// LS Electric XG5000 project: 0131 인버터 에스컬레이터
// PLC LSPLC

PROGRAM NewProgram (task: 스캔 프로그램)

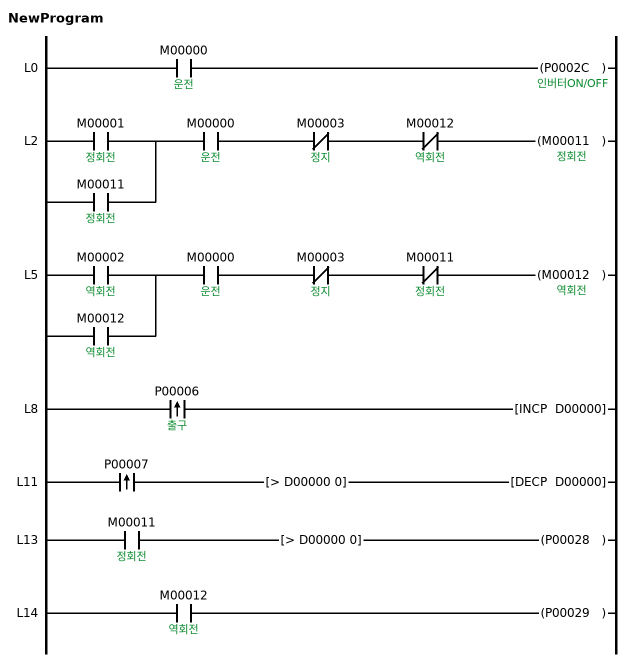
; L0
LOAD      M00000	// 운전
OUT       P0002C	// 인버터ON/OFF
; L2
LOAD      M00001	// 정회전
OR        M00011	// 정회전
AND       M00000	// 운전
AND NOT   M00003	// 정지
AND NOT   M00012	// 역회전
OUT       M00011	// 정회전
; L5
LOAD      M00002	// 역회전
OR        M00012	// 역회전
AND       M00000	// 운전
AND NOT   M00003	// 정지
AND NOT   M00011	// 정회전
OUT       M00012	// 역회전
; L8
LOADP     P00006	// 출구
INCP      D00000
; L11
LOADP     P00007
AND>      D00000 0
DECP      D00000
; L13
LOAD      M00011	// 정회전
AND>      D00000 0
OUT       P00028
; L14
LOAD      M00012	// 역회전
OUT       P00029